// TIA Portal project "Festo_Station 2_V15" (V15)

(* hardware
DEVICE "S7-1200-Station_1"  S7-1200 Station
   slot 0: "Baugruppenträger_0"  S7-1200 Rack  Rack  V1.0
   slot 1: "PLC_32"  CPU 1214C DC/DC/DC  6ES7 214-1AG31-0XB0  V3.0
   slot 3: "AQ 1x12BIT_1"  AQ1 signal board  6ES7 232-4HA30-0XB0  V1.0
*)

// ===== PLC "PLC_32"  CPU 1214C DC/DC/DC =====

VAR_GLOBAL   // PLC tag table "Standard-Variablentabelle"
   "System_Byte" AT %MB1 : Byte;
   "FirstScan" AT %M1.0 : Bool;
   "DiagStatusUpdate" AT %M1.1 : Bool;
   "AlwaysTRUE" AT %M1.2 : Bool;
   "AlwaysFALSE" AT %M1.3 : Bool;
   "Clock_Byte" AT %MB0 : Byte;
   "Clock_10Hz" AT %M0.0 : Bool;
   "Clock_5Hz" AT %M0.1 : Bool;
   "Clock_2.5Hz" AT %M0.2 : Bool;
   "Clock_2Hz" AT %M0.3 : Bool;
   "Clock_1.25Hz" AT %M0.4 : Bool;
   "Clock_1Hz" AT %M0.5 : Bool;
   "Clock_0.625Hz" AT %M0.6 : Bool;
   "Clock_0.5Hz" AT %M0.7 : Bool;
   "Part_AV" AT %I0.0 : Bool;   // Teil vorhanden
   "-2B1" AT %I0.7 : Bool;   // Zylinder2_eingefahren
   "-2B2" AT %I0.6 : Bool;   // Zylinder2_ausgefahren
   "-1B2" AT %I0.4 : Bool;   // Zylinder1_ausgefahren
   "-1B1" AT %I0.5 : Bool;   // Zylinder1_eingefahren
   "-1M1" AT %Q0.0 : Bool;   // Förderband
   "-B2" AT %I0.3 : Bool;   // Silber_Erkennung
   "-B3" AT %I0.2 : Bool;   // Rot_Erkennung
   "-B4" AT %I0.1 : Bool;   // Teil bei Rutsche_Voll
   "-1A1" AT %Q0.1 : Bool;   // Zylinder1_ausfahren
   "-2A1" AT %Q0.2 : Bool;   // Zinder2_ausfahren
   "-3A1" AT %Q0.3 : Bool;   // Stopper_einfahren
   "-S1" AT %I1.0 : Bool;   // Start
   "-S2" AT %I1.1 : Bool;   // Stopp
   "-S3" AT %I1.2 : Bool;   // Reset
END_VAR

DATA_BLOCK "Festo_Station_Sortierung_Kelmendi_DB"   // DB1
{ S7_Optimized_Access := 'TRUE' }
VERSION : 0.1
// stored: InstanceOfName Festo_Station_Sortierung_Kelmendi
"Festo_Station_Sortierung_Kelmendi"
BEGIN
END_DATA_BLOCK

FUNCTION_BLOCK "Festo_Station_Sortierung_Kelmendi"   // FB1, FBD
TITLE = Sortier_Station
{ S7_Optimized_Access := 'TRUE' }
VERSION : 0.1
   VAR_INPUT
      Start : Bool;
      Stopp : Bool;
      Reset : Bool;
      Teil_vorhanden : Bool;
      Silber_Sensor : Bool;
      Rot_Sensor : Bool;
      Rutsche_Sensor : Bool;
      Zylinder_Rot_ausgefahren : Bool;
      Zylinder_Silber_ausgefahren : Bool;
      Zylinder_Rot_eingefahren : Bool;
      Zylinder_Silber_eingefahren : Bool;
   END_VAR
   VAR_OUTPUT
      Motor_Förderband : Bool;
      Zylinder_Rot_ausfahren : Bool;
      Zylinder_Silber_ausfahren : Bool;
      Stopper_einfahren : Bool;
   END_VAR
   VAR
      freigabe : Bool;
      Grundstellung : Bool;
      "Schritt 1" : Bool;
      Silber_Teil : Bool;
      Rot_Teil : Bool;
      Schwarz_Teil : Bool;
      stopper_aus : Bool;
      Motor_aus : Bool;
      Teil_vorhanden_Timer : TOF_TIME;
      stopper_RS : Bool;
      Timer_schwarz : TON_TIME;
      Silber_Timer : TON_TIME;
      Rot_Timer : TON_TIME;
      Stopper_Timer : TOF_TIME;
      Impuls_Stopper : TP_TIME;
      Analyse_Zeit : TON_TIME;
      Hilfs_SR : Bool;
      Silber_Impuls : TP_TIME;
      Schwarz_Impuls : TP_TIME;
      Rot_Impuls : TP_TIME;
      Vereinzelungszeit : TP_TIME;
      "Rutsche_Rot_Auschalteverz." : TOF_TIME;
      Auschalteverz_Silber : TOF_TIME;
      "Auschalteverz._Schwarz" : TOF_TIME;
      Schwarz_Timer : TON_TIME;
      Rot_Wartezeit : TON_TIME;
   END_VAR
BEGIN

REGION Network 1: Freigabe
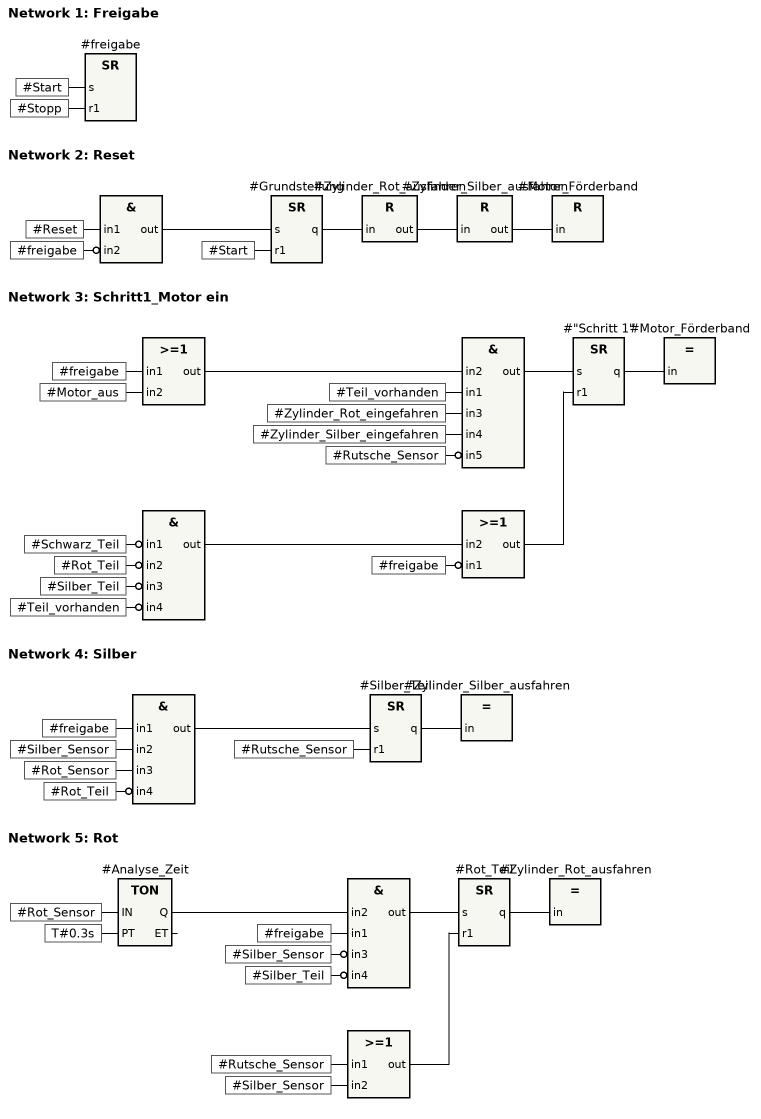
   IF #Start THEN
       #freigabe := TRUE;   // SR flip-flop
   END_IF;
   IF #Stopp THEN #freigabe := FALSE; END_IF;
END_REGION

REGION Network 2: Reset
   IF #Reset AND NOT #freigabe THEN
       #Grundstellung := TRUE;   // SR flip-flop
   END_IF;
   IF #Start THEN #Grundstellung := FALSE; END_IF;
   IF #Grundstellung THEN
       #Zylinder_Rot_ausfahren := FALSE;
       #Zylinder_Silber_ausfahren := FALSE;
       #Motor_Förderband := FALSE;
   END_IF;
END_REGION

REGION Network 3: Schritt1_Motor ein
   IF (#freigabe OR #Motor_aus) AND #Teil_vorhanden AND #Zylinder_Rot_eingefahren AND #Zylinder_Silber_eingefahren AND NOT #Rutsche_Sensor THEN
       #"Schritt 1" := TRUE;   // SR flip-flop
   END_IF;
   IF (NOT #Schwarz_Teil AND NOT #Rot_Teil AND NOT #Silber_Teil AND NOT #Teil_vorhanden) OR NOT #freigabe THEN
       #"Schritt 1" := FALSE;
   END_IF;
   #Motor_Förderband := #"Schritt 1";
END_REGION

REGION Network 4: Silber
   IF #freigabe AND #Silber_Sensor AND #Rot_Sensor AND NOT #Rot_Teil THEN
       #Silber_Teil := TRUE;   // SR flip-flop
   END_IF;
   IF #Rutsche_Sensor THEN #Silber_Teil := FALSE; END_IF;
   #Zylinder_Silber_ausfahren := #Silber_Teil;
END_REGION

REGION Network 5: Rot
   #Analyse_Zeit(IN := #Rot_Sensor, PT := T#0.3s);   // TON
   IF #Analyse_Zeit.Q AND #freigabe AND NOT #Silber_Sensor AND NOT #Silber_Teil THEN
       #Rot_Teil := TRUE;   // SR flip-flop
   END_IF;
   IF #Rutsche_Sensor OR #Silber_Sensor THEN #Rot_Teil := FALSE; END_IF;
   #Zylinder_Rot_ausfahren := #Rot_Teil;
END_REGION

REGION Network 6: Schwarz
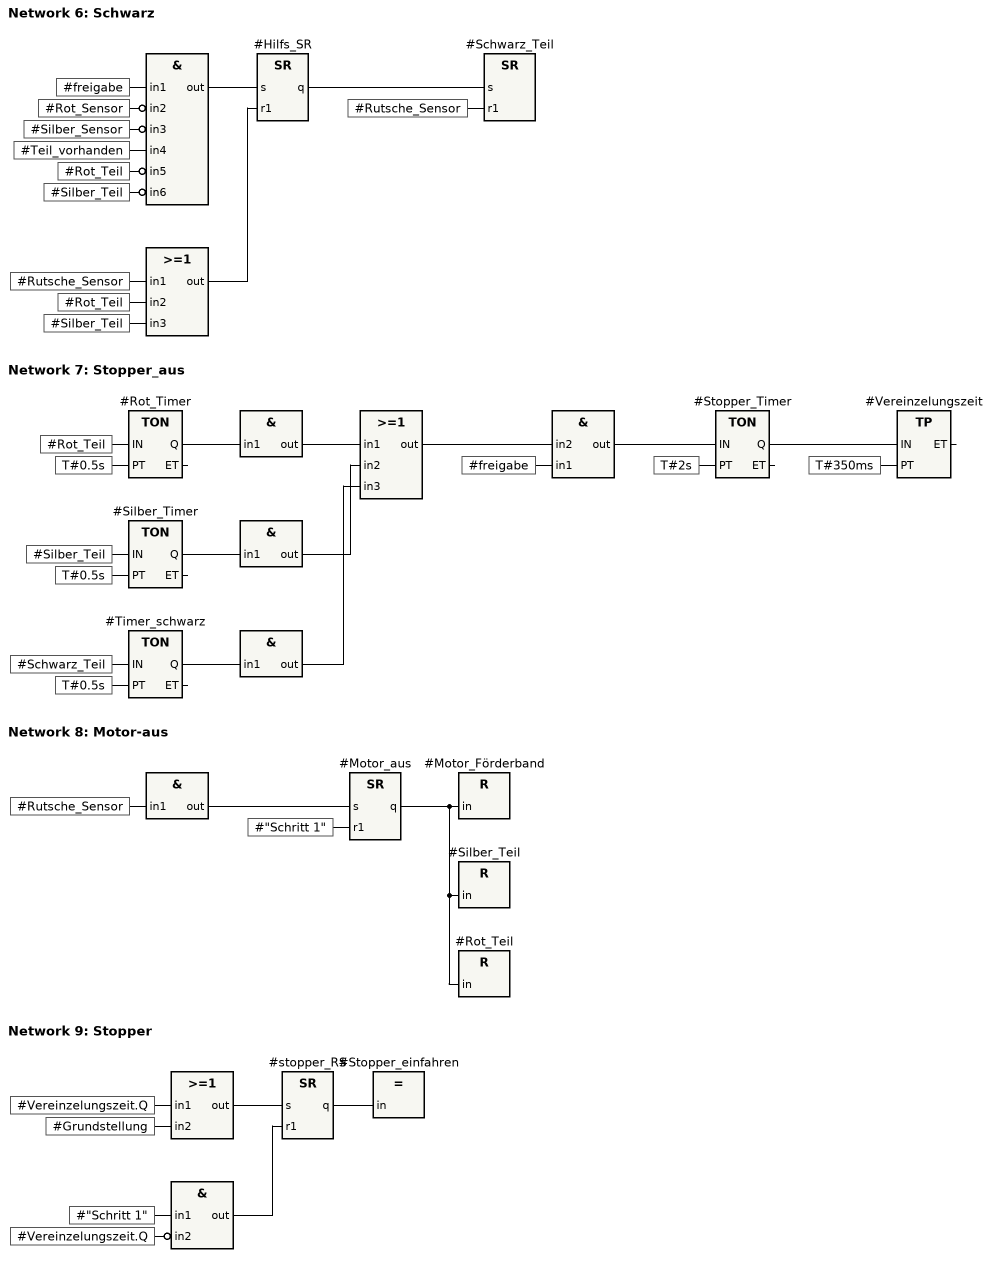
   IF #freigabe AND NOT #Rot_Sensor AND NOT #Silber_Sensor AND #Teil_vorhanden AND NOT #Rot_Teil AND NOT #Silber_Teil THEN
       #Hilfs_SR := TRUE;   // SR flip-flop
   END_IF;
   IF #Rutsche_Sensor OR #Rot_Teil OR #Silber_Teil THEN #Hilfs_SR := FALSE; END_IF;
   IF #Hilfs_SR THEN
       #Schwarz_Teil := TRUE;   // SR flip-flop
   END_IF;
   IF #Rutsche_Sensor THEN #Schwarz_Teil := FALSE; END_IF;
END_REGION

REGION Network 7: Stopper_aus
   #Rot_Timer(IN := #Rot_Teil, PT := T#0.5s);   // TON
   #Silber_Timer(IN := #Silber_Teil, PT := T#0.5s);   // TON
   #Timer_schwarz(IN := #Schwarz_Teil, PT := T#0.5s);   // TON
   #Stopper_Timer(IN := (#Rot_Timer.Q OR #Silber_Timer.Q OR #Timer_schwarz.Q) AND #freigabe, PT := T#2s);   // TON
   #Vereinzelungszeit(IN := #Stopper_Timer.Q, PT := T#350ms);   // TP
END_REGION

REGION Network 8: Motor-aus
   IF #Rutsche_Sensor THEN
       #Motor_aus := TRUE;   // SR flip-flop
   END_IF;
   IF #"Schritt 1" THEN #Motor_aus := FALSE; END_IF;
   IF #Motor_aus THEN
       #Motor_Förderband := FALSE;
       #Silber_Teil := FALSE;
       #Rot_Teil := FALSE;
   END_IF;
END_REGION

REGION Network 9: Stopper
   IF #Vereinzelungszeit.Q OR #Grundstellung THEN
       #stopper_RS := TRUE;   // SR flip-flop
   END_IF;
   IF #"Schritt 1" AND NOT #Vereinzelungszeit.Q THEN #stopper_RS := FALSE; END_IF;
   #Stopper_einfahren := #stopper_RS;
END_REGION
END_FUNCTION_BLOCK

ORGANIZATION_BLOCK "Main"   // OB1, FBD, ProgramCycle
TITLE = "Main Program Sweep (Cycle)"
{ S7_Optimized_Access := 'TRUE' }
VERSION : 0.1
BEGIN

REGION Network 1: Sortierung_station
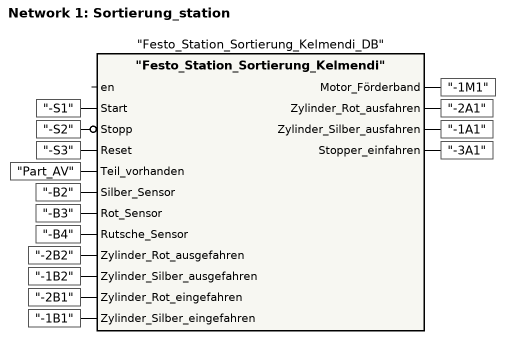
   "Festo_Station_Sortierung_Kelmendi_DB"(Start := "-S1",   // "Festo_Station_Sortierung_Kelmendi"
                           Stopp := NOT "-S2",
                           Reset := "-S3",
                           Teil_vorhanden := "Part_AV",
                           Silber_Sensor := "-B2",
                           Rot_Sensor := "-B3",
                           Rutsche_Sensor := "-B4",
                           Zylinder_Rot_ausgefahren := "-2B2",
                           Zylinder_Silber_ausgefahren := "-1B2",
                           Zylinder_Rot_eingefahren := "-2B1",
                           Zylinder_Silber_eingefahren := "-1B1",
                           Motor_Förderband => "-1M1",
                           Zylinder_Rot_ausfahren => "-2A1",
                           Zylinder_Silber_ausfahren => "-1A1",
                           Stopper_einfahren => "-3A1");
END_REGION
END_ORGANIZATION_BLOCK